// TIA Portal V17 export
// export: Created 2022-07-20T07:02:39.5923685Z, ExportSetting WithDefaults, DisplayName Totally Integrated Automation Portal, DisplayVersion V17, DisplayName TIA Portal Openness, DisplayVersion V17, DisplayName TIA Portal Version Control Interface, DisplayVersion V17, DisplayName SINAMICS Startdrive Advanced, DisplayVersion V17, DisplayName SINAMICS Startdrive G130, G150, S120, S150, SINAMICS MV, S210, DisplayVersion V17, DisplayName SINAMICS Startdrive G110M, G120, G120C, G120D, G120P, G115D, DisplayVersion V17, DisplayName STEP 7 Professional, DisplayVersion V17, DisplayName STEP 7 Safety, DisplayVersion V17, DisplayName WinCC Advanced, DisplayVersion V17
VAR_GLOBAL   // PLC tag table "LCalcMC_ErrorIDs"
END_VAR
VAR_GLOBAL CONSTANT   // user constants
   LCALCMC_ERR_ACCEL_INVALID : Word := 16#8201;
   LCALCMC_ERR_DECEL_INVALID : Word := 16#8202;
   LCALCMC_ERR_DISTANCE_INVALID : Word := 16#8203;
   LCALCMC_ERR_JERK_INVALID : Word := 16#8204;
   LCALCMC_ERR_TIME_INVALID : Word := 16#8206;
   LCALCMC_ERR_VELOCITY_INVALID : Word := 16#8207;
   LCALCMC_ERR_NEGATIVE_RESULT : Word := 16#8401;
   LCALCMC_ERR_JERK_OUT_OF_BOUNDS : Word := 16#8403;
   LCALCMC_ERR_NOT_SOLVABLE : Word := 16#8404;
   LCALCMC_ERR_VELOCITY_OUT_OF_BOUNDS : Word := 16#8405;
   LCALCMC_ERR_ACCEL_OUT_OF_BOUNDS : Word := 16#8406;
   LCALCMC_ERR_DECEL_OUT_OF_BOUNDS : Word := 16#8407;
   LCALCMC_ERR_NO_ZERO_FOUND : Word := 16#8408;
   LCALCMC_ERR_REVERSAL_NOT_ALLOWED : Word := 16#8205;
   LCALCMC_ERR_DISTANCE_SIGN_WRONG : Word := 16#8209;
   LCALCMC_ERR_POLY_LESS_THAN_3RD_DEGREE : Word := 16#8208;
   LCALCMC_ERR_TIME_OUT_OF_BOUNDS : Word := 16#8409;
   LCALCMC_ERR_TIME_DECREASE_ACCEL_TOO_SMALL : Word := 16#8402;
END_VAR
